(* Logix 5000 project; controller PLC2_Project_7_SensorCalibration Emulate 5570 rev 20.11; software revision 20.00 *)

TASK MainTask (continuous, watchdog 500 ms) : MainProgram

MODULES
   Local : Emulate 5570 (ICP 1, rev 20.11)
END_MODULES

ADD_ON_INSTRUCTION NSCP   (* revision 1.0 *)
// Nicks Scale With Parameters
VAR_INPUT
   InputMax : DINT; {required}
   InputMin : DINT; {required}
   ScaledMaxOut : DINT; {required}
   ScaledMinOut : DINT; {required}
   Input : DINT; {required}
END_VAR
VAR_OUTPUT
   ScaledOutput : REAL; {access Read Only, required}
END_VAR
VAR
   Rate : REAL; {access None}
END_VAR

ROUTINE Logic   (* structured text *)
   IF (EnableIn) THEN
   	Rate := (ScaledMaxOut - ScaledMinOut) / (InputMax - InputMin);
   	ScaledOutput := (Input - InputMin) * Rate + ScaledMinOut;
   END_IF;
END_ROUTINE
END_ADD_ON_INSTRUCTION

ADD_ON_INSTRUCTION SCP   (* revision 1.2, vendor Rockwell Automation *)
// Scale w/Parameters
// Help:
// Use this instruction to scale data from your analog module and bring it into the limits prescribed by the process variable or another analog module.
// Equations used in calculating a linear relationship:
// Scaled value = (input value - input min.) x rate + scaled minimum
// Rate = (scaled max. - scaled min.) / (input max. - input min.)
VAR_INPUT
   Input : REAL; {required}
   Input_Min : REAL; {required}
   Input_Max : REAL; {required}
   Scaled_Min : REAL; {required}
   Scaled_Max : REAL; {required}
END_VAR
VAR_OUTPUT
   Output : REAL; {access Read Only, required}
END_VAR
VAR
   Rate : REAL;
END_VAR

ROUTINE Logic   (* ladder *)
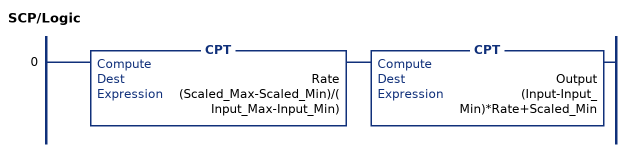
   0: CPT(Rate,(Scaled_Max-Scaled_Min)/(Input_Max-Input_Min))CPT(Output,(Input-Input_Min)*Rate+Scaled_Min);
END_ROUTINE
END_ADD_ON_INSTRUCTION

PROGRAM MainProgram   (* main routine _00_MainRoutine *)
VAR
   _NSCP_O2SensorOutput : NSCP; {access Read Only}
   _ONS_calibrate : BOOL; {access Read Only}
   _ONS_calibrationComplete : BOOL; {access Read Only}
   _ONS_CalibrationStartBit : BOOL; {access Read Only}
   _ONS_off : BOOL; {access Read Only}
   _ONS_sampling : BOOL; {access Read Only}
   _sim_outputSensor : REAL; {access Read Only}
   _sim_oxygenGasValveInput : BOOL; {access Read Only}
   _sim_timer : TIMER; {access Read Only}
   _sim_zeroGasValveInput : BOOL; {access Read Only}
   Button_Auto : BOOL; {access Read Only}
   Button_CalibrateMode : BOOL; {access Read Only}
   Button_SampleMode : BOOL; {access Read Only}
   Calibrate_Seq0_Delay_Timer : TIMER := (PRE := 2000); {access Read Only}
   Calibrate_Seq0_Timer : TIMER := (PRE := 30000); {access Read Only}
   Calibrate_Seq1_Delay_Timer : TIMER := (PRE := 2000); {access Read Only}
   Calibrate_Seq1_Timer : TIMER := (PRE := 30000); {access Read Only}
   Calibration_Complete : BOOL; {access Read Only}
   Calibration_Seq : DINT; {access Read Only}   // Calibration Sequence: 0 - Waiting 1 - Test nuetral gas 2 - Test oxy gas 3 - Calibrate sensor
   Calibration_StartSeqBit : BOOL; {access Read Only}
   Gas_Neutral_Average : REAL; {access Read Only}
   Gas_Neutral_SampleCount : COUNTER; {access Read Only}
   Gas_Neutral_TotalSample : DINT; {access Read Only}
   Gas_Test_Average : REAL; {access Read Only}
   Gas_Test_SampleCount : COUNTER; {access Read Only}
   Gas_Test_TotalSample : DINT; {access Read Only}
   O2sensor_MaxRawInput : DINT; {access Read Only}
   O2sensor_RawReading : DINT; {access Read Only}
   O2Sensor_ScaledReading : REAL; {access Read Only}
   OneSecond_Timer_1 : TIMER := (PRE := 1000); {access Read Only}
   OneSecond_Timer_2 : TIMER := (PRE := 1000); {access Read Only}
   System_Mode : DINT := 2; {access Read Only}   // 0 = Sample Mode 1 = Calibrate Mode 2 = Off
   System_SamplingMode_Timer : TIMER := (PRE := 60000); {access Read Only}   // The time to continuously measure the air O2 level
   Valve_TestGas_En : BOOL; {access Read Only}
   Valve_ZeroGas_En : BOOL; {access Read Only}
END_VAR

ROUTINE _00_MainRoutine   (* ladder *)
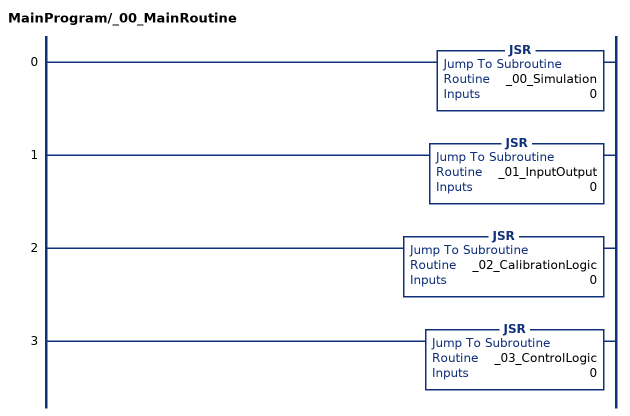
   0: JSR(_00_Simulation,0);
   1: JSR(_01_InputOutput,0);
   2: JSR(_02_CalibrationLogic,0);
   3: JSR(_03_ControlLogic,0);
END_ROUTINE

ROUTINE _00_Simulation   (* structured text *)
// Simulates the external system for our project. Responds to inputs, produces outputs
   // Analog output simulation
   // Range:
   // 0 - 16383
   // 0% - 40%
   
   IF(_sim_zeroGasValveInput)THEN
   	_sim_outputSensor := 0; // 0 - 16384
   END_IF;
   
   IF(_sim_oxygenGasValveInput)THEN
   	_sim_outputSensor := 12287; //12287 =~ 30% gas
   	//_sim_outputSensor := 9999; // Test value. After calibration, output should still read ~ 30%
   	//Change this value (lower) to see if the calibration works
   END_IF;
   
   //Decrease the sensor output over time to represent the sensor degrading:
   
   
   
END_ROUTINE

ROUTINE _01_InputOutput   (* ladder *)
// Fake inputs and outputs from and to simulation
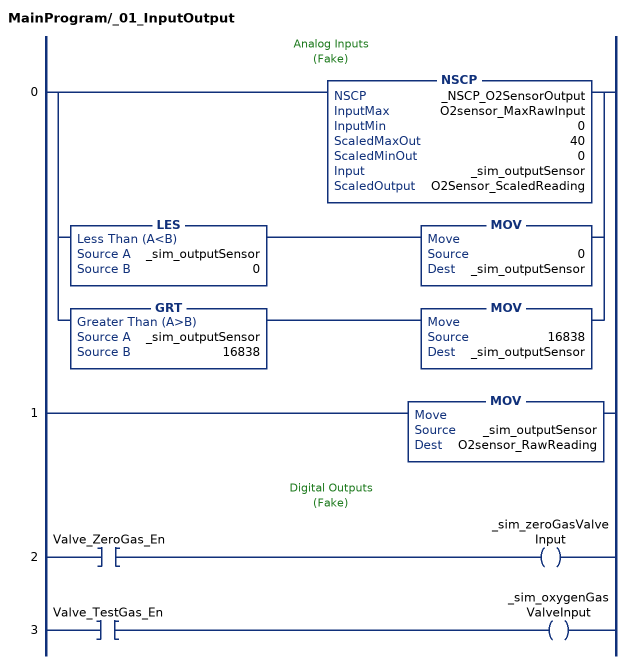
   // Analog Inputs
   // (Fake)
   0: [NSCP(_NSCP_O2SensorOutput,O2sensor_MaxRawInput,0,40,0,_sim_outputSensor,O2Sensor_ScaledReading) ,LES(_sim_outputSensor,0) MOV(0,_sim_outputSensor) ,GRT(_sim_outputSensor,16838) MOV(16838,_sim_outputSensor) ];
   1: MOV(_sim_outputSensor,O2sensor_RawReading);
   // Digital Outputs
   // (Fake)
   2: XIC(Valve_ZeroGas_En)OTE(_sim_zeroGasValveInput);
   3: XIC(Valve_TestGas_En)OTE(_sim_oxygenGasValveInput);
END_ROUTINE

ROUTINE _02_CalibrationLogic   (* ladder *)
// Logic for O2 Sensor calibration sequence
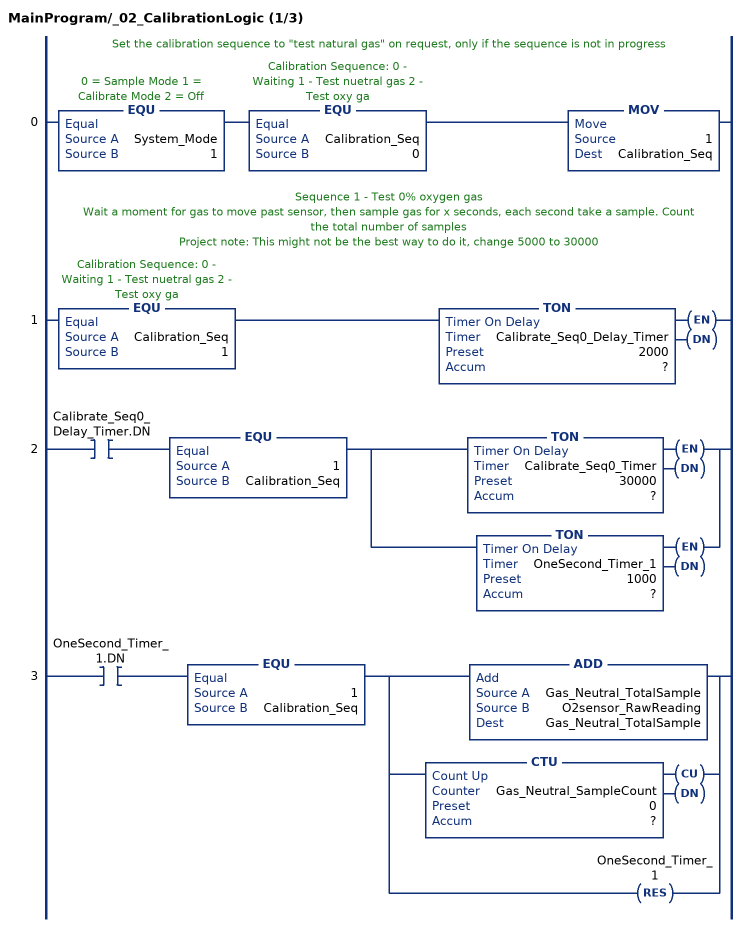
   // Set the calibration sequence to "test natural gas" on request, only if the sequence is not in progress
   0: EQU(System_Mode,1)EQU(Calibration_Seq,0)MOV(1,Calibration_Seq);
   // Sequence 1 - Test 0% oxygen gas
   // Wait a moment for gas to move past sensor, then sample gas for x seconds, each second take a sample. Count the total number of samples
   // Project note: This might not be the best way to do it, change 5000 to 30000
   1: EQU(Calibration_Seq,1)TON(Calibrate_Seq0_Delay_Timer,?,?);
   2: XIC(Calibrate_Seq0_Delay_Timer.DN)EQU(1,Calibration_Seq)[TON(Calibrate_Seq0_Timer,?,?) ,TON(OneSecond_Timer_1,?,?) ];
   3: XIC(OneSecond_Timer_1.DN)EQU(1,Calibration_Seq)[ADD(Gas_Neutral_TotalSample,O2sensor_RawReading,Gas_Neutral_TotalSample) ,CTU(Gas_Neutral_SampleCount,?,?) ,RES(OneSecond_Timer_1) ];
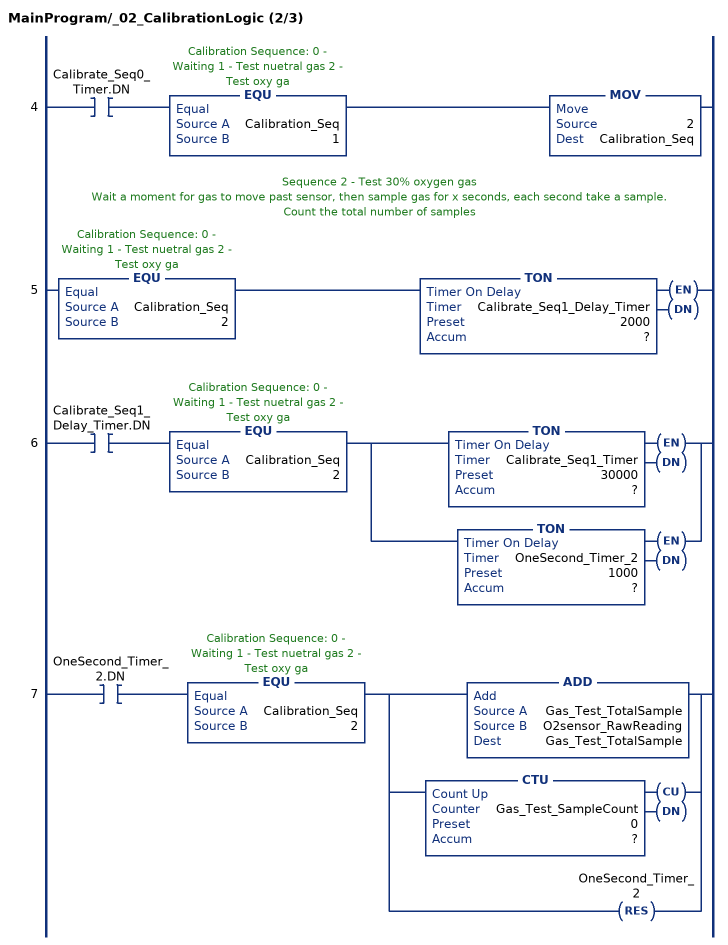
   4: XIC(Calibrate_Seq0_Timer.DN)EQU(Calibration_Seq,1)MOV(2,Calibration_Seq);
   // Sequence 2 - Test 30% oxygen gas
   // Wait a moment for gas to move past sensor, then sample gas for x seconds, each second take a sample. Count the total number of samples
   5: EQU(Calibration_Seq,2)TON(Calibrate_Seq1_Delay_Timer,?,?);
   6: XIC(Calibrate_Seq1_Delay_Timer.DN)EQU(Calibration_Seq,2)[TON(Calibrate_Seq1_Timer,?,?) ,TON(OneSecond_Timer_2,?,?) ];
   7: XIC(OneSecond_Timer_2.DN)EQU(Calibration_Seq,2)[ADD(Gas_Test_TotalSample,O2sensor_RawReading,Gas_Test_TotalSample) ,CTU(Gas_Test_SampleCount,?,?) ,RES(OneSecond_Timer_2) ];
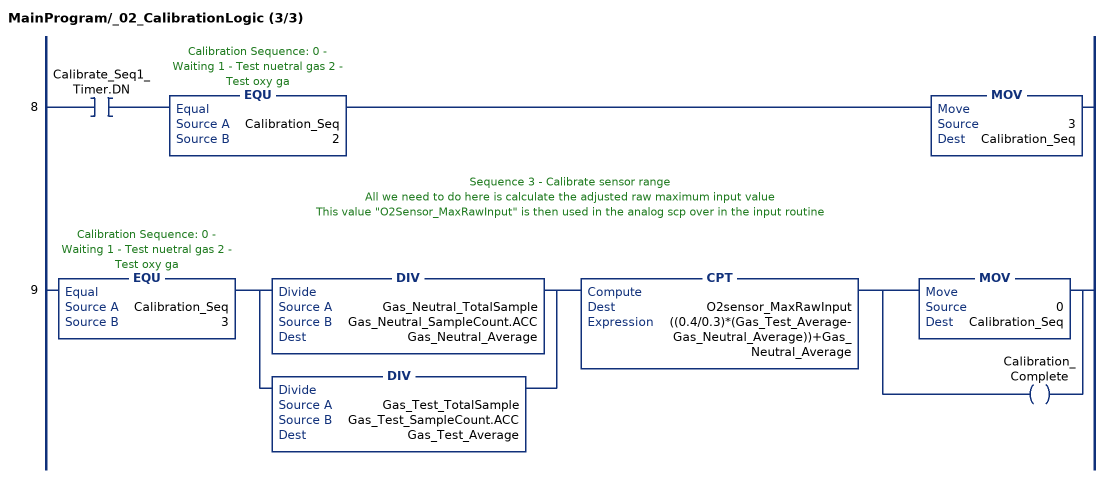
   8: XIC(Calibrate_Seq1_Timer.DN)EQU(Calibration_Seq,2)MOV(3,Calibration_Seq);
   // Sequence 3 - Calibrate sensor range
   // All we need to do here is calculate the adjusted raw maximum input value
   // This value "O2Sensor_MaxRawInput" is then used in the analog scp over in the input routine
   9: EQU(Calibration_Seq,3)[DIV(Gas_Neutral_TotalSample,Gas_Neutral_SampleCount.ACC,Gas_Neutral_Average) ,DIV(Gas_Test_TotalSample,Gas_Test_SampleCount.ACC,Gas_Test_Average) ]CPT(O2sensor_MaxRawInput,((0.4/0.3)*(Gas_Test_Average-Gas_Neutral_Average))+Gas_Neutral_Average)[MOV(0,Calibration_Seq) ,OTE(Calibration_Complete) ];
END_ROUTINE

ROUTINE _03_ControlLogic   (* ladder *)
// 02 Sensor controller. Switches between sampling & calibration
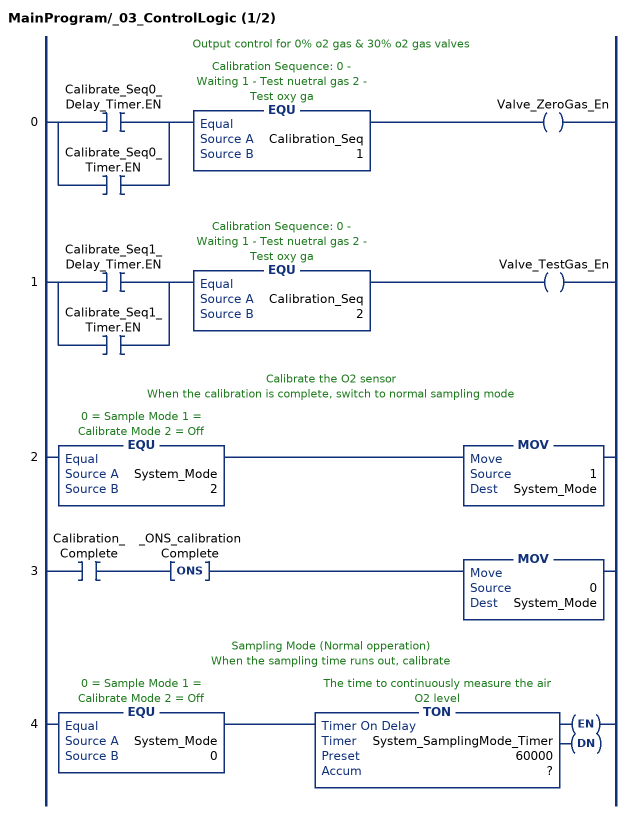
   // Output control for 0% o2 gas & 30% o2 gas valves
   0: [XIC(Calibrate_Seq0_Delay_Timer.EN) ,XIC(Calibrate_Seq0_Timer.EN) ]EQU(Calibration_Seq,1)OTE(Valve_ZeroGas_En);
   1: [XIC(Calibrate_Seq1_Delay_Timer.EN) ,XIC(Calibrate_Seq1_Timer.EN) ]EQU(Calibration_Seq,2)OTE(Valve_TestGas_En);
   // Calibrate the O2 sensor
   // When the calibration is complete, switch to normal sampling mode
   2: EQU(System_Mode,2)MOV(1,System_Mode);
   3: XIC(Calibration_Complete)ONS(_ONS_calibrationComplete)MOV(0,System_Mode);
   // Sampling Mode (Normal opperation)
   // When the sampling time runs out, calibrate
   4: EQU(System_Mode,0)TON(System_SamplingMode_Timer,?,?);
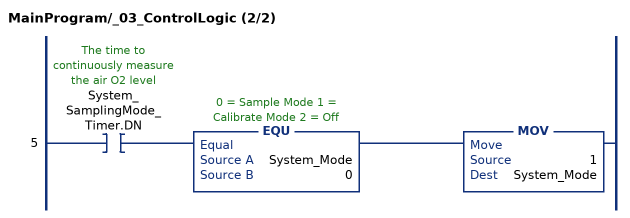
   5: XIC(System_SamplingMode_Timer.DN)EQU(System_Mode,0)MOV(1,System_Mode);
END_ROUTINE
END_PROGRAM
